PROGRAM MAIN
VAR
	eState : E_MachineState;
	bStart : BOOL;
	bLimitUp : BOOL;
	bLimitDown : BOOL;
	bEmergencyStop : BOOL;
	bDrilling : BOOL;
	bRetracting : BOOL;
	
	
END_VAR


IF bEmergencyStop THEN
	 eState := E_MachineState.Error;
END_IF

CASE eState OF
	E_MachineState.IDLE :
	bDrilling := FALSE;
	bRetracting := FALSE;
	IF MAIN.TRANS_DrillCheck THEN
		eState := E_MachineState.Drilling;
	END_IF
	
	E_MachineState.Drilling :
	bDrilling := TRUE;
	bRetracting := FALSE;
	bLimitUp := FALSE;
	IF bStart AND bLimitDown THEN
		eState := E_MachineState.Retracting;
	END_IF
	
	E_MachineState.Retracting :
	bDrilling := FALSE;
	bRetracting := TRUE;
	bLimitDown := FALSE;
	IF bStart AND bLimitUp THEN
		eState := E_MachineState.IDLE;
	END_IF
	
	E_MachineState.Error :
	bDrilling := FALSE;
	bRetracting := FALSE;
	IF  NOT bEmergencyStop AND bStart THEN
		eState := E_MachineState.IDLE;
	END_IF
	
	
END_CASE

TRANSITION TRANS_DrillCheck:
TRANS_DrillCheck := (bStart AND bLimitUp);
END_TRANSITION

END_PROGRAM

(* stored: Version 1.1.0.1, ProductVersion 3.1.4024.16
   POU MAIN: Id {24e244ad-bb03-43f3-8a06-f0ff732d53b2}, SpecialFunc None
   Transition TRANS_DrillCheck: Id {4ca51243-dbe5-483e-bebb-ad8ff64c1c2c} *)
